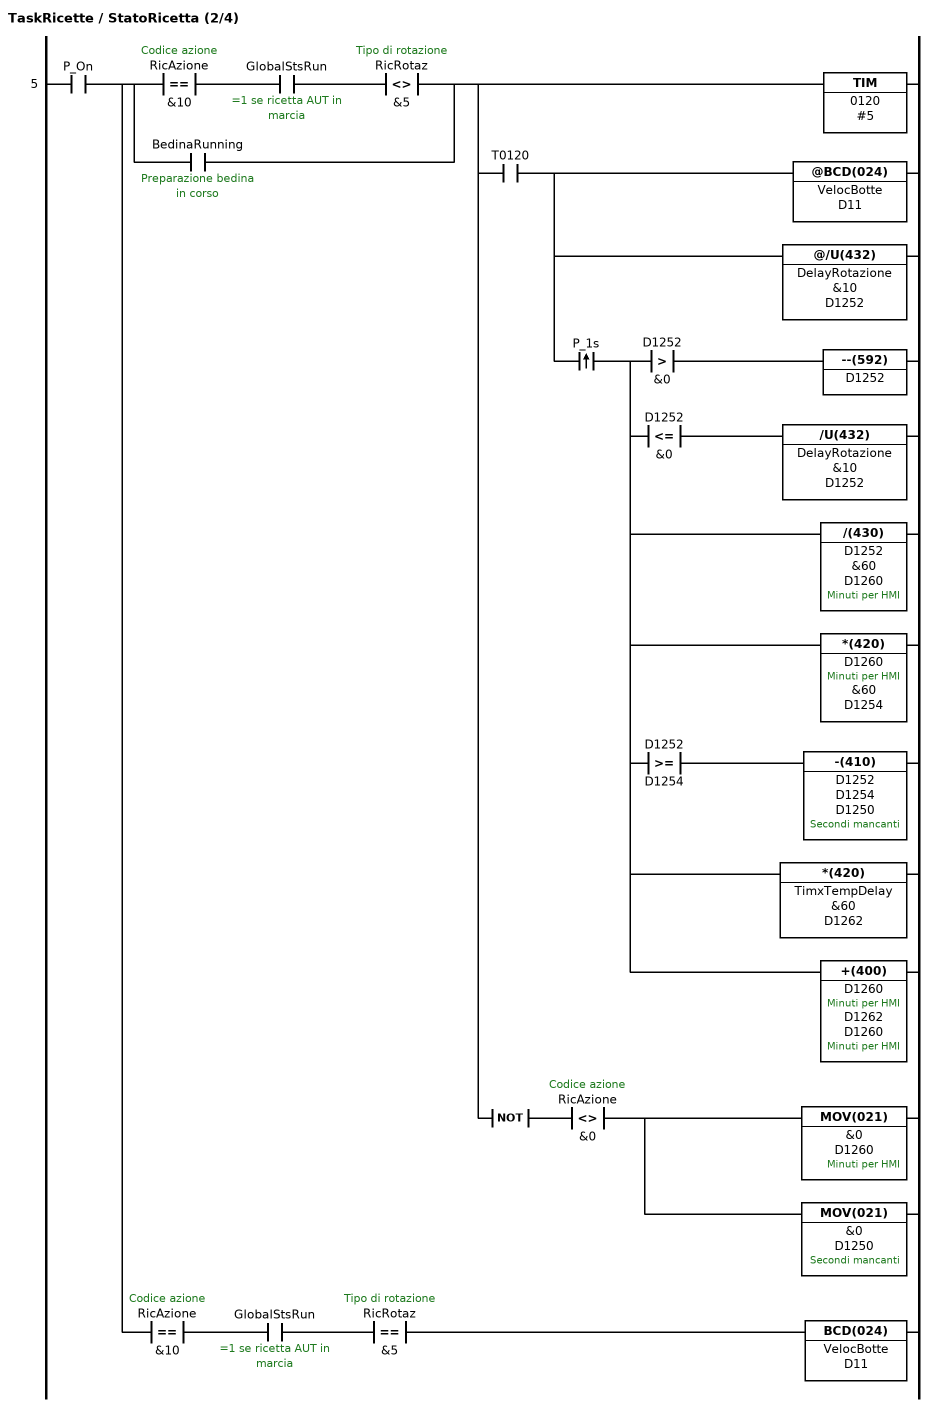
; [picture p48: TaskRicette / StatoRicetta, rungs 5-5]
; rung 5
LD P_On
OUT TR0
LD=(300) RicAzione &10  ; Codice azione
AND GlobalStsRun  ; =1 se ricetta AUT in marcia
AND<>(305) RicRotaz &5  ; Tipo di rotazione
OR BedinaRunning  ; Preparazione bedina in corso
ANDLD
OUT TR1
TIM 0120 #5
AND T0120
@BCD(024) VelocBotte D11
@/U(432) DelayRotazione &10 D1252
@AND P_1s
OUT TR2
AND>(320) D1252 &0
--(592) D1252
LD TR2
AND<=(315) D1252 &0
/U(432) DelayRotazione &10 D1252
LD TR2
/(430) D1252 &60 D1260  ; Minuti per HMI
*(420) D1260 &60 D1254  ; Minuti per HMI
AND>=(325) D1252 D1254
-(410) D1252 D1254 D1250  ; Secondi mancanti
LD TR2
*(420) TimxTempDelay &60 D1262
+(400) D1260 D1262 D1260  ; Minuti per HMI
LD TR1
NOT(520)
AND<>(305) RicAzione &0  ; Codice azione
MOV(021) &0 D1260  ; Minuti per HMI
MOV(021) &0 D1250  ; Secondi mancanti
LD TR0
AND=(300) RicAzione &10  ; Codice azione
AND GlobalStsRun  ; =1 se ricetta AUT in marcia
AND=(300) RicRotaz &5  ; Tipo di rotazione
BCD(024) VelocBotte D11

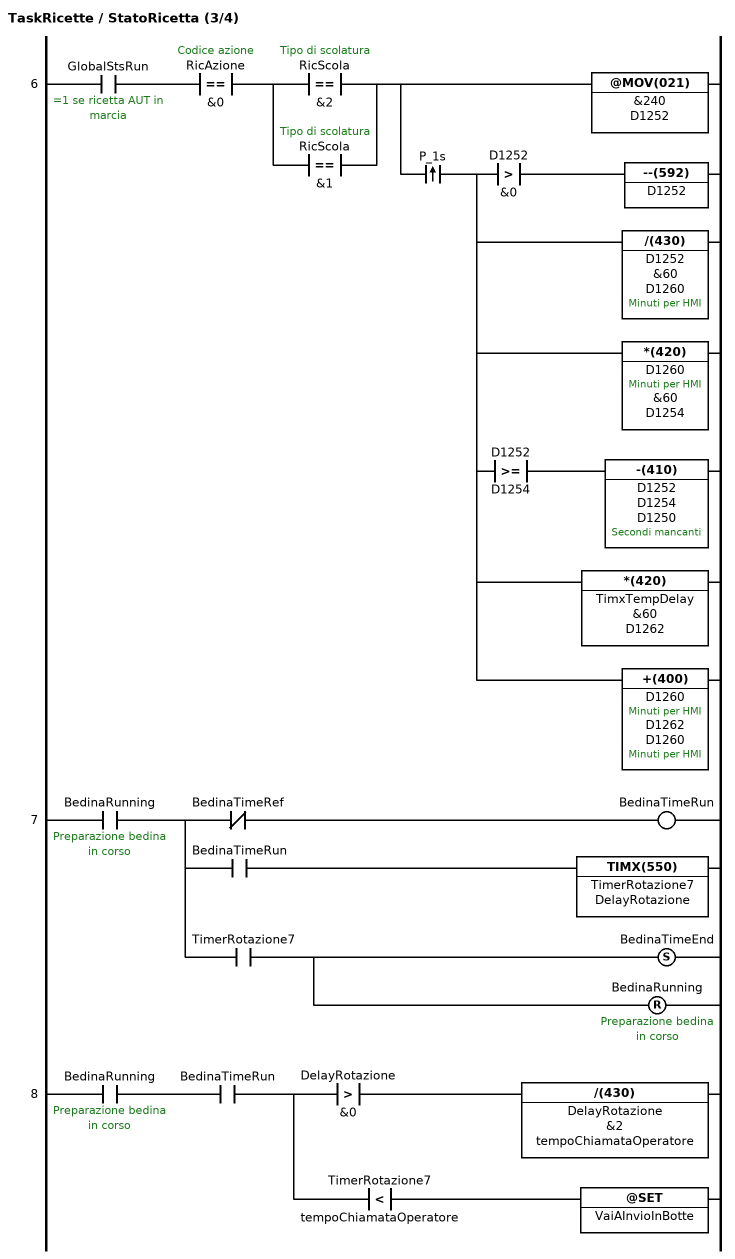
; rung 6
LD GlobalStsRun  ; =1 se ricetta AUT in marcia
AND=(300) RicAzione &0  ; Codice azione
LD=(300) RicScola &2  ; Tipo di scolatura
OR=(300) RicScola &1  ; Tipo di scolatura
ANDLD
@MOV(021) &240 D1252
@AND P_1s
OUT TR0
AND>(320) D1252 &0
--(592) D1252
LD TR0
/(430) D1252 &60 D1260  ; Minuti per HMI
*(420) D1260 &60 D1254  ; Minuti per HMI
AND>=(325) D1252 D1254
-(410) D1252 D1254 D1250  ; Secondi mancanti
LD TR0
*(420) TimxTempDelay &60 D1262
+(400) D1260 D1262 D1260  ; Minuti per HMI
; rung 7
LD BedinaRunning  ; Preparazione bedina in corso
OUT TR0
ANDNOT BedinaTimeRef
OUT BedinaTimeRun
LD TR0
AND BedinaTimeRun
TIMX(550) TimerRotazione7 DelayRotazione
LD TR0
AND TimerRotazione7
SET BedinaTimeEnd
RSET BedinaRunning  ; Preparazione bedina in corso
; rung 8
LD BedinaRunning  ; Preparazione bedina in corso
AND BedinaTimeRun
OUT TR0
AND>(320) DelayRotazione &0
/(430) DelayRotazione &2 tempoChiamataOperatore
LD TR0
AND<(310) TimerRotazione7 tempoChiamataOperatore
@SET VaiAInvioInBotte

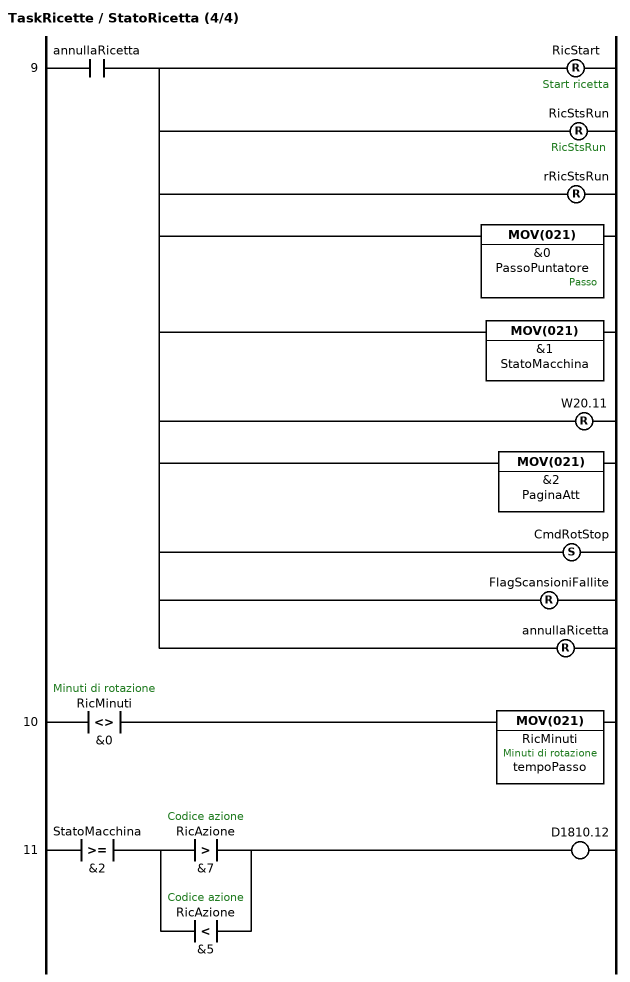
; rung 9
LD annullaRicetta
RSET RicStart  ; Start ricetta
RSET RicStsRun  ; RicStsRun
RSET rRicStsRun
MOV(021) &0 PassoPuntatore  ; Passo
MOV(021) &1 StatoMacchina
RSET W20.11
MOV(021) &2 PaginaAtt
SET CmdRotStop
RSET FlagScansioniFallite
RSET annullaRicetta
; rung 10
LD<>(305) RicMinuti &0  ; Minuti di rotazione
MOV(021) RicMinuti tempoPasso  ; Minuti di rotazione
; rung 11
LD>=(325) StatoMacchina &2
LD>(320) RicAzione &7  ; Codice azione
OR<(310) RicAzione &5  ; Codice azione
ANDLD
OUT D1810.12

### Section END

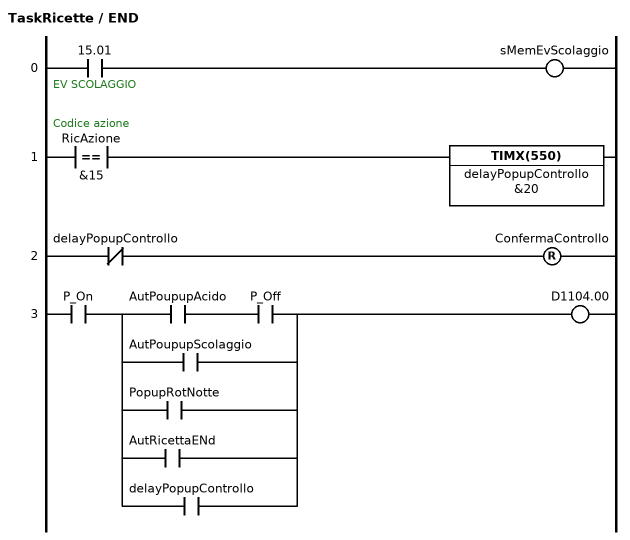
; rung 0
LD 15.01  ; EV SCOLAGGIO
OUT sMemEvScolaggio
; rung 1
LD=(300) RicAzione &15  ; Codice azione
TIMX(550) delayPopupControllo &20
; rung 2
LDNOT delayPopupControllo
RSET ConfermaControllo
; rung 3
LD P_On
LD AutPoupupAcido
AND P_Off
OR AutPoupupScolaggio
OR PopupRotNotte
OR AutRicettaENd
OR delayPopupControllo
ANDLD
OUT D1104.00
; rung 4
END(001)

## Program CicliStep (cyclic task 2)
Local symbols
CmdRst D2000.00 BOOL
CmdStart D2000.01 BOOL
Index D2010 INT
MemRiga D2012 WORD
StepCiclo D2001.00 BOOL[15]
StsEnd D2000.02 BOOL
StsRun D2000.03 BOOL
TempAnnoNecessario D2016 DINT
i D2014 INT
reset1 W20.10 BOOL
reset2 W20.11 BOOL
tempCondStep1 W20.12 BOOL
 IF TimerSaltaPasso.CF = TRUE  AND MemTimSkip=FALSE THEN
	Index:= 1;
	CmdRotAv:= false;
	CmdRotInd:= false;
	CmdRotAlt:= false;
	CmdRotStop:= false;
	CmdRotNotte:= false;
	CmdAcqua:= false;
	CmdFormico:= false;
	CmdGlutaral:= false;
	CmdScolaggioDecrementoAsse:= false;
	CmdScolaggioNormale:= false;
	PopupMancatoScolaggio:= false;
	RichiestaLetturaBarcode:= false;
	AutCmdNotturno:= false;
	AutPoupupScolaggio:= false;

end_if;
MemTimSkip:= TimerSaltaPasso.CF;
 
 (*Stop Riga*)
IF NOT  RicStart then
	StsRun:= false;
	(*StsEnd:= true;
	Index:= 5;*)
END_IF;
 
 
 (* Reset ciclo e comandi vari *)
IF CmdRst = TRUE THEN
	StsRun:= false;
	CmdStart:= false;
	CmdRst := false;	
END_IF;
GlobalGreenFlash:= false;
GlobalGreenLight:= false;
LetturaPesoREAL:= DINT_TO_REAL(LetturaPesoDINT);
		LetturaPesoREAL:= LetturaPesoREAL/1000,0;
		TolleranzaInf:= PesoNecessarioRicetta-((PesoNecessarioRicetta*Tolleranza)/100,0);
	(*I comandi da temperatura sono SET, vengono resettati dopo 1s sennò non li prende usando il momentaneo*)
TIMX(CmdTemperaturaON=true,TimerPIDon,10);
TIMX(CmdTemperaturaOFF=true,TimerPIDoff,10);
IF TimerPIDon.CF=TRUE THEN
	CmdTemperaturaON:= false;
END_IF;
IF TimerPIDoff.CF=TRUE THEN
	CmdTemperaturaOFF:= false;
END_IF;
(*Salvataggio ID riga per cambio riga*)
IF RicRigNum<>MemRiga THEN
	CmdStart:= true;
END_IF;
MemRiga:= RicRigNum;

(* Start riga *)
IF (CmdStart AND RicStsRun)= true THEN
	StsRun:= true;
	Index:= 1;
	CmdStart:= false;
	StsEnd:= false;
	FlagStsEnd:= false;
ELSIF RicStsRun=FALSE THEN
	StsRun:= false;
	Index:= 0;
END_IF;

FOR i:=0 TO 5 DO
	IF Index=i THEN	
		StepCiclo[i]:= true;
	ELSE
		StepCiclo[i]:= false;
	END_if;
END_FOR;

(* Cicli in base a codice azione *)
(* RIempimento acqua *)
IF RicAzione=5 THEN
	(* Passaggio parametri *)
	IF StepCiclo[1]=true THEN
		TemperaturaAcquaPerBCD:= INT_TO_WORD(((WORD_TO_INT(RicGradi)) * 10));
		LitriAcqua:= INT_TO_BCD_WORD(REAL_TO_INT(RicPeso/10,0));
		(*Controllo se è già stato eseguito un riempimento in precedenza*)
		IF FlagRiempimentoAcqua = TRUE THEN
			(*Riempimento già eseguito, richiedo la presenza operatore*)
			PopupMancatoScolaggio:= TRUE;
			IF PopupMancatoScolaggio=TRUE AND ConfermaMancatoScolaggio THEN (*Quando viene confermato il riempimento nonostante non ho scolaggio*)
				PopupMancatoScolaggio:= false;
				ConfermaMancatoScolaggio:= false;
				Index:= 2;
			END_IF;
		ELSE (*Se non è già avvenuto, proseguo*)		
			Index:= 2;
		end_if;
	END_IF;
	(*Comando*)
	IF StepCiclo[2]=true THEN
		CmdAcqua:= true;
		Index:= 3;
	END_IF;
	(* Attesa ritorno *)
	IF StepCiclo[3]=TRUE AND (FeedbackAcqua=TRUE OR (acqua_litriErogati >= (acqua_setpointRicetta/2))) THEN
		FlagRiempimentoAcqua:= TRUE;
		Index:= 4;
	END_IF;
	(* Attesa fine operazione *)
	(*IF StepCiclo[4]=true AND FeedbackAcqua=false THEN*)
	IF StepCiclo[4]=true AND (FeedbackAcqua=false OR (acqua_litriErogati >= (acqua_setpointRicetta/2)))  THEN
		TemperaturaMacchina:= TemperaturaAcqua;
		VelocBotte:= 9;
		CmdTemperaturaON:= true;
		IF NOT flagPrimoRiempimento then
			CmdRotAv:= true;
			IF FeedbackRotAv=TRUE then
				CmdRotAv:= FALSE;
				flagPrimoRiempimento := true;
				StsRun:= false;
				StsEnd:= true;			
			end_if;
		ELSIF flagPrimoRiempimento THEN
			StsRun:= false;
			StsEnd:= true;	
		end_if;		
	END_IF;
END_IF;

(* RIempimento formico *)
IF RicAzione=6 THEN
	(* Passaggio parametri *)
	tempCondStep1:= StepCiclo[1]=true  AND presenzaOpAcido=FALSE AND VaiAInvioInBotte=TRUE;
	TIMX(tempCondStep1,TimerFormico1,20);
	TIMX(TimerFormico1.CF,TimerFormico2,40);
	TIMX(StepCiclo[2]=true,TimerFormico3,20);
	TIMX(StepCiclo[2]=true,TimerFormico4,40);
	TIMX(StepCiclo[3]=true,TimerFormico5,20);
	TIMX(StepCiclo[3]=true,TimerFormico6,40);
	IF StepCiclo[1]=true THEN
		AutPoupupTBedina:= 1;
		PesoFormico:=  INT_TO_BCD_WORD(REAL_TO_INT(RicPeso*10,0));
		(*AutPoupupAcido:= TRUE;
		IF presenzaOpAcido=TRUE THEN
			presenzaOpAcido:= FALSE;*)
		IF VaiAInvioInBotte=TRUE AND presenzaOpAcido=FALSE THEN															(*attesa metà rotazione*)
			RichiestaFormico:= true;
			IF TimerFormico1.CF=TRUE THEN
				RichiestaFormico:= false;
				IF TimerFormico2.CF=TRUE THEN
					Index:= 2;
				END_IF;
			END_IF;
		END_IF;
	end_if;
	(*Comando*)
	IF StepCiclo[2]=true THEN
		SceltaFormico:= true;
		IF TimerFormico3.CF=TRUE THEN
			SceltaFormico:= false;
			IF TimerFormico4.CF=TRUE THEN
			Index:= 3;
			END_IF;
		END_IF;
	END_IF;
	(* Attesa ritorno *)
	IF StepCiclo[3] =true THEN
		CmdFormico:= true;
		IF TimerFormico5.CF=TRUE THEN
			CmdFormico:= false;
			
			IF TimerFormico6.CF=TRUE AND FeedbackFormico=TRUE THEN
				(*AutPoupupAcido:= true;
				confermaVaiABedina:= true;
				Index:= 4;*)
				Index:= 5;
			END_IF;
				END_IF;
	END_IF;
	(* Attesa fine operazione *)
	IF StepCiclo[4]=true AND AutPoupupAcido=false AND FeedbackFormico=false THEN
		AutPoupupTBedina:= 0;
		confermaVaiABedina:= false;
		IF confermaVaiABedina=FALSE then
			StsRun:= false;
			StsEnd:= true;
		end_if;
	END_IF;
	IF StepCiclo[5]=TRUE AND FeedbackFormico=false THEN
		AutPoupupAcido:= true;
		confermaVaiABedina:= true;
		IF AutPoupupAcido = TRUE then
			Index := 4;
		end_if;
	end_if;
	IF StepCiclo[4] = TRUE OR StepCiclo[5] = TRUE THEN
		visualizzaKgAcido := TRUE;
	ELSE
		visualizzaKgAcido:= FALSE;
	end_If;
END_IF;

(* RIempimento glutaraldeide *)
IF RicAzione=7 THEN
	(* Passaggio parametri *)
	TIMX(StepCiclo[1]=true,TimerGlutar1,20);
	TIMX(StepCiclo[1]=true,TimerGlutar2,40);
	TIMX(StepCiclo[2]=true,TimerGlutar3,20);
	TIMX(StepCiclo[2]=true,TimerGlutar4,40);
	TIMX(StepCiclo[3]=true,TimerGlutar5,20);
	TIMX(StepCiclo[3]=true,TimerGlutar6,40);
	IF StepCiclo[1]=true THEN
		AutPoupupTBedina:= 1;
		PesoGlutaral:=  INT_TO_BCD_WORD(REAL_TO_INT(RicPeso*10,0));
		AutPoupupAcido:= TRUE;
		IF presenzaOpAcido=TRUE THEN
			presenzaOpAcido:= FALSE;
			SceltaGlutar:= true;
			IF TimerGlutar1.CF=TRUE THEN
				SceltaGlutar:= false;
				IF TimerGlutar2.CF=TRUE THEN
					Index:= 2;
				END_IF;
			END_IF;
		end_if;
	END_IF;
	(*Comando*)
	IF StepCiclo[2]=true THEN
		RichiestaGlutar:= true;
		IF TimerGlutar3.CF=TRUE THEN
			RichiestaGlutar:= false;
			IF TimerGlutar4.CF=TRUE THEN
			Index:= 3;
			END_IF;
		END_IF;
	END_IF;
	(* Attesa ritorno *)
	IF StepCiclo[3] =true THEN
		CmdGlutaral:= true;
		IF TimerGlutar5.CF=TRUE THEN
			CmdGlutaral:= false;
			IF TimerGlutar6.CF=TRUE AND FeedbackGlutaral=TRUE THEN
				(*AutPoupupAcido:= true;
				Index:= 4;*)
				Index:= 5;
			END_IF;
				END_IF;
	END_IF;
	(* Attesa fine operazione *)
	IF StepCiclo[4]=true AND AutPoupupAcido=false AND FeedbackGlutaral=false THEN
		AutPoupupTBedina:= 0;
		confermaVaiABedina:= false;
		IF confermaVaiABedina=FALSE THEN
			StsRun:= false;
			StsEnd:= true;
		end_if;
	END_IF;
	IF StepCiclo[5]=TRUE AND FeedbackFormico=FALSE THEN
		AutPoupupAcido:=TRUE;
		confermaVaiABedina:=TRUE;
		IF AutPoupupAcido=TRUE THEN
			Index:= 4;
		end_if;
	END_IF;
	
	IF StepCiclo[4]=TRUE OR StepCiclo[5]=TRUE THEN
		visualizzaKgGlutaral:= TRUE;
	ELSE
		visualizzaKgGlutaral:= FALSE;
	END_IF;
END_IF;

(* Aggiorna temperatura macchina in rotazione *)
IF RicAzione=10 THEN
	IF RicGradi <> 0 then
		TemperaturaMacchina :=  INT_TO_BCD_WORD(((WORD_TO_INT(RicGradi)) * 10));
	ELSE
		TemperaturaMacchina := 10;
	end_if;
end_if;


(* Rotazione avanti, tipo 1 *)
IF RicAzione=10 AND RicRotaz=1 THEN
	(* Passaggio parametri *)
	IF StepCiclo[1]=true THEN
		VelocBotte:= INT_TO_WORD(REAL_TO_INT((INT_TO_REAL(WORD_TO_INT(RicSpeed))) * 1,24));
		Index:= 2;
	END_IF;
	(*Comando*)
	IF StepCiclo[2]=true THEN
		CmdRotAv:= true;
		Index:= 3;
	END_IF;
	(* Attesa ritorno *)
	IF StepCiclo[3]=true AND FeedbackRotAv=true THEN
		TIMX(StepCiclo[3]=true,TimerRotazione,DelayRotazione);
		CmdRotAv:= false;
		IF TimerRotazione.CF THEN		
			Index:= 4;
		END_IF;
	END_IF;
	(* Attesa fine operazione *)
	IF StepCiclo[4]=true  THEN	
		StsRun:= false;
		StsEnd:= true;
	END_IF;
END_IF;

(* Rotazione indietro, tipo 2 *)
IF RicAzione=10 AND RicRotaz=2 THEN
	(* Passaggio parametri *)
	IF StepCiclo[1]=true THEN
		VelocBotte:= INT_TO_WORD(REAL_TO_INT((INT_TO_REAL(WORD_TO_INT(RicSpeed))) * 1,24));
		Index:= 2;
	END_IF;
	(*Comando*)
	IF StepCiclo[2]=true THEN
		CmdRotInd:= true;
		Index:= 3;
	END_IF;
	(* Attesa ritorno *)
	IF StepCiclo[3]=true AND FeedbackRotInd=true THEN
		TIMX(StepCiclo[3]=true,TimerRotazione,DelayRotazione);
		CmdRotInd:= false;
		IF TimerRotazione.CF THEN		
			Index:= 4;
		END_IF;
	END_IF;
	(* Attesa fine operazione *)
	IF StepCiclo[4]=true  THEN	
		StsRun:= false;
		StsEnd:= true;
	END_IF;
END_IF;

(* Rotazione alternata, tipo 3 *)
IF RicAzione=10 AND RicRotaz=3 THEN
	(* Passaggio parametri *)
	IF StepCiclo[1]=true THEN
		VelocBotte:= INT_TO_WORD(REAL_TO_INT((INT_TO_REAL(WORD_TO_INT(RicSpeed))) * 1,24));
		IF RicMinuti<=60 then
			DelayRotazione:= (WORD_TO_UINT(RicMinuti)*600);
			TimxTempDelay:= 0;
		ELSIF RicMinuti>60 THEN
			TimxTempDelay:= 0;
			TimxRicMinuti:= WORD_TO_INT(RicMinuti);
			WHILE TimxRicMinuti>60 DO
				TimxRicMinuti:= TimxRicMinuti-60;
				TimxTempDelay:= TimxTempDelay+1;
			END_WHILE;
			DelayRotazione:= (INT_TO_UINT(TimxRicMinuti))*600;
		end_if;
		Index:= 2;
		CmdRotAlt:= true;
	END_IF;
	(*Comando*)
	TIMX(StepCiclo[2]=TRUE,timerRotazioneStep2, 10);
	IF StepCiclo[2]=true AND timerRotazioneStep2.CF = TRUE THEN
		Index:= 3;
	END_IF;
	(* Attesa ritorno *)
	IF TimxTempDelay= 0 then
		TIMX(StepCiclo[3]=true,TimerRotazione3,DelayRotazione);
	ELSIF TimxTempDelay>0 THEN
		TIMX(StepCiclo[3]=true,TimerRotazione3,36000);
	end_if;
	IF StepCiclo[3]=true AND FeedbackRotAlt=true THEN
		CmdRotAlt:= false;
		IF TimerRotazione3.CF THEN
				IF TimxTempDelay= 0 then
					Index:= 4;
				ELSIF TimxTempDelay>0 THEN
					TimxTempDelay:=TimxTempDelay-1;
					Index:= 2;
				end_if;
		END_IF;
	END_IF;
	(* Attesa fine operazione *)
	IF StepCiclo[4]=true  THEN	
		StsRun:= false;
		StsEnd:= true;
	END_IF;
END_IF;

(* Ferma rotazione, tipo 4 *)
IF RicAzione=10 AND RicRotaz=4 THEN
	(* Passaggio parametri *)
	IF StepCiclo[1]=true THEN
		Index:= 2;
	END_IF;
	(*Comando*)
	IF StepCiclo[2]=true THEN
		CmdRotStop:= true;
		Index:= 3;
	END_IF;
	(* Attesa ritorno *)
	TIMX(StepCiclo[3]=true,TimerRotazione4,100);
	IF StepCiclo[3]=true THEN
		IF TimerRotazione4.CF THEN		
			CmdRotStop:= FALSE;
			Index:= 4;
		END_IF;
	END_IF;
	(* Attesa fine operazione *)
	IF StepCiclo[4]=true  THEN	
		StsRun:= false;
		StsEnd:= true;
	END_IF;
END_IF;

(* Rotazione alternata notte, tipo 5 *)
IF RicAzione=10 AND RicRotaz=5 THEN
	(* Passaggio parametri *)
	IF StepCiclo[1]=true THEN
		PopupRotNotte:= false;
		VelocBotte:= 6;
		OreAltPreNotte:= 0;
		MinAltPreNotte:= 5;
		Index:= 2;
	END_IF;
	(*Comando*)
	IF StepCiclo[2]=true THEN
		AutCmdNotturno:= TRUE;
		Index:= 3;
	END_IF;
	(* Attesa ritorno *)
	IF StepCiclo[3]=true AND FeedbackRotAlt=true THEN
			PopupRotNotte:= true;
			Index:= 4;
		END_IF;
	END_IF;
	(* Attesa fine operazione *)
	IF StepCiclo[4]=true AND ConfermaRotNotte=true  THEN
		PopupRotNotte:= false;
		StsRun:= false;
		StsEnd:= true;
	END_IF;

(* Rotazione alternata, tipo 7 *)
IF RicAzione=10 AND RicRotaz=7 THEN
	(* Passaggio parametri *)
	IF StepCiclo[1]=true THEN
		BedinaTimeEnd:= FALSE;
		VelocBotte:= INT_TO_WORD(REAL_TO_INT((INT_TO_REAL(WORD_TO_INT(RicSpeed))) * 1,24));
		IF RicMinuti<=60 then
			DelayRotazione:= (WORD_TO_UINT(RicMinuti)*600);
			TimxBedinaDelay:= 0;
		ELSIF RicMinuti>60 THEN
			TimxBedinaDelay:= 0;
			TimxRicMinuti:= WORD_TO_INT(RicMinuti);
			WHILE TimxRicMinuti>60 DO
				TimxRicMinuti:= TimxRicMinuti-60;
				TimxBedinaDelay:= TimxBedinaDelay+1;
			END_WHILE;
			DelayRotazione:= (INT_TO_UINT(TimxRicMinuti))*600;
		end_if;
		Index:= 2;
		CmdRotAlt:= true;
		BedinaRunning:= true;
	END_IF;
	(*Comando*)
	IF StepCiclo[2]=true THEN
		Index:= 3;
	END_IF;
	
	IF StepCiclo[3]=true AND FeedbackRotAlt=true THEN
		CmdRotAlt:= false;
		AutPupupInvioBotte:= FALSE;
	    Index:= 4;
	END_IF;
	(* Attesa fine operazione *)
	IF StepCiclo[4]=true  THEN	
		StsRun:= false;
		StsEnd:= true;
		(*BedinaRunning:= FALSE;*)
	END_IF;
END_IF;

(* Preparazione bedina, tipo 7  *)
IF RicAzione=50 AND RicRotaz=7 THEN
	(* Passaggio parametri *)
	IF StepCiclo[1]=true THEN
		(*VaiAInvioInBotte:= TRUE;*)
		RichiestaLetturaBarcode:= TRUE;
		AutPoupupBedina:= 1;
		AutPoupupTBedina:= 1;
		FlagAbilitaScansioni:= TRUE;
	        	
				FlagScansioniFallite:= FALSE;
				FlagIgnoraScansioniFallite:= FALSE;
				NumeroScansioni:= 0;
				FlagRitentaScansioni:= FALSE;
				StatoScansione:= 0;
		Index:= 2;
	END_IF;
	(*Comando*)
	IF StepCiclo[2]=true AND ((LetturaPesoREAL=0,0) AND LetturaCodPro=0 AND LetturaRicetta=0) THEN
		ProdottoErratoPopup:= false;
		StatoScansione:= 1;
		Index:= 3;
	END_IF;
	(* Attesa ritorno *)

	IF StepCiclo[3]=true AND (FlagScansioniFallite=FALSE) AND (LetturaPesoREAL<>0,0) AND (LetturaCodPro<>0) AND (LetturaRicetta<>0) THEN
		(*Conversione peso da DINT da bilanca a reale, in Kg. Calcolo tolleranze da parametro tolleranza % (5%, per ora)*)
		LetturaPesoREAL:= DINT_TO_REAL(LetturaPesoDINT);
		LetturaPesoREAL:= LetturaPesoREAL/REAL1000;
		TolleranzaInf:= PesoNecessarioRicetta-((PesoNecessarioRicetta*Tolleranza)/PercentualeREAL);
		TolleranzaSup:= PesoNecessarioRicetta+((PesoNecessarioRicetta*Tolleranza)/PercentualeREAL);
		(*Su codice a barre Anno e n°Ricetta sono un codice unico, vengono uniti in quanto separati*)
		TempAnnoNecessario:= INT_TO_DINT(AnnoNecessarioRicetta);
		LetturaRicettaTemp:= (TempAnnoNecessario*10000000)+(RicettaNecessariaRicetta);
		
						
		(*Controlla corrispondeza peso, codice prodotto, codice ricetta*)
			IF LetturaPesoREAL>TolleranzaInf AND LetturaPesoREAL<TolleranzaSup AND LetturaCodPro= CodiceNecessarioRicetta AND LetturaRicetta=LetturaRicettaTemp then		
				Index:= 4;
				FlagNuovaScansione:= false;
				RichiestaLetturaBarcode:= FALSE;
				AutPoupupBedina:= 0;
				AutPoupupTBedina:= 0;
				FlagAbilitaScansioni:= FALSE;
				NumeroScansioni:= 0;
				ELSE
				(*Se il prodotto non è giusto, segno 1 tentativo e resetto tutto*)
				StatoScansione:= 2;
				
				IF NumeroScansioni<2 THEN
					NumeroScansioni:= NumeroScansioni+1;
					Index:= 2;
				
				ELSIF NumeroScansioni>=2 THEN
					FlagScansioniFallite:= TRUE;
									
				END_IF;;
		
		FlagNascondiTasti:= NOT(FlagScansioniFallite OR RichiestaLetturaBarcode);
	END_IF;
				
END_IF;		
	(* Attesa fine operazione *)
		IF StepCiclo[3]=true AND FlagScansioniFallite=TRUE THEN
			AutPoupupBedina:= 0;
			IF FlagIgnoraScansioniFallite=TRUE THEN
				FlagScansioniFallite:= FALSE;
				FlagIgnoraScansioniFallite:= FALSE;
				RichiestaLetturaBarcode:= FALSE;
			    AutPoupupBedina:= 0;
				NumeroScansioni:= 0;
				Index:= 4;
			END_IF;
		END_IF;		
	(*invio in bedina manuale completato, conferma da operatore*)
	IF StepCiclo[4]=true  THEN
		
		ConfermaBedina:= False;
		RichiestaConfermaBedina:= false;
		StsRun:= false;
		StsEnd:= true;
				
	END_IF;
END_IF;

(* Invio in botte, tipo 8 *)
IF RicAzione=10 AND RicRotaz=8 THEN
	IF StepCiclo[1]=true AND BedinaTimeEnd=FALSE THEN
	AutPoupupTBedina:= 1;
	END_IF;
	(* Passaggio parametri *)
	IF StepCiclo[1]=true AND BedinaTimeEnd=TRUE THEN
		IF FlagSolido=TRUE THEN
			CmdRotStop:= true;
		end_if;
		Index:= 2;
		AutPoupupTBedina:= 0;
		BedinaTimeEnd:= FALSE;
	END_IF;
	(*Comando*)
	TIMX(StepCiclo[2]=true,TimerRotazione4,100);
	IF StepCiclo[2]=true THEN
		IF FlagSolido=TRUE THEN
			IF TimerRotazione4.CF THEN		
				CmdRotStop:= FALSE;
				Index:= 3;
				FlagSolido:= false;
				(*VaiAInvioInBotte:= true;*)
			END_IF;
		ELSE
			Index:= 3;
			(*VaiAInvioInBotte:= true;*)
		end_if;
	END_IF;
	(* Attesa ritorno *)
	IF StepCiclo[3]=true THEN
		AutPupupInvioBotte:= true;
			Index:= 4;
		(*END_IF;*)
	END_IF;
	(* Attesa fine operazione *)
	IF invioConRisciacquoON OR invioSenzaRisciacquoON THEN
		ConfermaInvioBotte:= FALSE;
	end_if;
	IF StepCiclo[4]=true AND ConfermaInvioBotte=true AND NOT invioConRisciacquoON AND NOT invioSenzaRisciacquoON THEN	
		ConfermaInvioBotte:= false;
		AutPupupInvioBotte:= false;
		StsRun:= false;
		StsEnd:= true;
	END_IF;
END_IF;

(* Controllo *)
IF RicAzione=15 THEN
	(* Passaggio parametri *)
	IF StepCiclo[1]=true THEN
		Index:= 2;
	END_IF;
	(*Comando*)
	IF StepCiclo[2]=true THEN
		Index:= 3;
	END_IF;
	(* Attesa ritorno *)
	IF StepCiclo[3]=true AND delayPopupControllo.CF=TRUE THEN
		Index:= 4;
	END_IF;
	(* Attesa fine operazione *)
	IF StepCiclo[4]=true AND ConfermaControllo=True AND delayPopupControllo.CF=TRUE THEN	
		ConfermaControllo:= false;
		StsRun:= false;
		StsEnd:= true;
	END_IF;
END_IF;

(*Scolaggio a decremento da asse*)
IF RicScola=2 AND RicAzione= 0 THEN
	IF StepCiclo[1]=TRUE THEN
		CmdScolaggioDecrementoAsse:= true;
		IF StsScolaggioDecrementoAsse=TRUE THEN
			CmdScolaggioDecrementoAsse:= false;
			Index:= 2;
		END_IF;
	END_IF;
	IF StepCiclo[2]=TRUE THEN
		IF AutCmdStop=TRUE THEN
			FlagRiempimentoAcqua:= false;
			StsRun:= false;
			StsEnd:= true;
			flagPrimoRiempimento :=  FALSE;
		END_IF;
	END_IF;
(*ELSIF RicScola=1 AND RicAzione= 0 THEN
	IF StepCiclo[1]=TRUE THEN
		CmdScolaggioNormale:= true;
		TIMX(StepCiclo[1],TimerScolaggioON,10);
		IF TimerScolaggioON.CF=TRUE THEN
			CmdScolaggioNormale:= false;
			Index:= 2;
		END_IF;
	END_IF;
	IF StepCiclo[2]=TRUE THEN
		IF StsScolaggioNormale=FALSE THEN
			StsRun:= false;
			StsEnd:= true;
		END_IF;
	END_IF;*)
IF RicScola<>0 OR RicAzione=99 then
	CmdTemperaturaOFF:= true;
	TemperaturaMacchina:= 1;
end_if;
END_IF;	
TIMX((RicScola=1),TimerScolaggioNormale,2400);
IF RicScola=1 AND RicAzione= 0 THEN	
	IF TimerScolaggioNormale.CF = TRUE AND NOT flagFineScolaggio THEN
		AutPoupupScolaggio:= TRUE;
		flagFineScolaggio:= TRUE;
	END_IF;
	IF StepCiclo[1]=TRUE THEN
		CmdScolaggioNormale:= true;
		IF StsScolaggioNormale=TRUE THEN
			CmdScolaggioNormale:= false;
			Index:= 2;
		END_IF;
	END_IF;
	IF StepCiclo[2]=TRUE THEN
		IF AutCmdStop=TRUE THEN
			FlagRiempimentoAcqua:= false;
			StsRun:= false;
			StsEnd:= true;
			flagFineScolaggio:= FALSE;
			flagPrimoRiempimento :=  FALSE;
		END_IF;
	END_IF;
END_IF;	
(*Con la pausa non incremento il passo a fine azione*)
IF (NOT RicPause) AND RicStart then
	(* Cambio riga su fronte dello status end. Aumenta il puntatore e carica il passo successivo*)
	IF StsEnd<>FlagStsEnd THEN
		RicStato:=2;
		PassoPuntatoreINT:= WORD_TO_INT(PassoPuntatore);
		PassoPuntatoreINT:= (PassoPuntatoreINT+1);
		PassoPuntatore:= INT_TO_WORD(PassoPuntatoreINT);
		CaricaRIcetta:= true;
	END_IF;
	FlagStsEnd:= StsEnd;
ELSE
	StsRun:= false;
END_IF;

	
(*Copia  stsRun e comandi torretta luminosa in variabili globali*)
GlobalStsRun:= StsRun;
(*Se sono in marcia automatica, controllo torretta e stati in automatico, altrimenti sono esclusi*)
IF StsRun=TRUE then
	IF RicAzione=50 OR RicAzione=10 OR RicAzione=15 then
		CASE WORD_TO_INT(RicRotaz) OF
			1..7: (*Con rotazioni standard, luce fissa*)
				GlobalGreenLight:= true;
			(*7: Se invio in bedina o in botte, la luce lampeggia
				GlobalGreenFlash:= true;*)
		END_CASE;
	END_IF;
	(*Lampeggio torretta con conferma di mancato scolaggio*)
	IF (RicAzione=5 AND PopupMancatoScolaggio=TRUE) OR (RicAzione=10 AND  RicRotaz=8 AND BedinaRunning=FALSE) OR (RicAzione=15) (*OR (RicAzione=6)*)OR AutPoupupScolaggio= TRUE OR RicScola = 1 OR confermaVaiABedina=TRUE OR inserimentoProdottiRunning OR VaiAInvioInBotte THEN
		GlobalGreenFlash:= TRUE;
	END_IF;
    IF (RicAzione=10 AND  RicRotaz=8 AND BedinaRunning=TRUE) OR (RicAzione=0 AND RicScola=2 AND PopupMancatoScolaggio=false AND AutPoupupScolaggio= FALSE)  THEN
		GlobalGreenLight:= TRUE;
	END_IF;
	reset1:= FALSE;
ELSE
	(*Lo StsRun si reinizializza su ogni passo, attenzione alle memorie che vengono inserite di seguito*)
	(*Resetta memoria usate dalla ricetta*)
	IF reset1=FALSE then
	GlobalGreenLight:= false;
	GlobalGreenFlash:= false;
	RicAzione:= 0;
	RicRotaz:= 0;
	VisibilitàIndietroMan:= true;
	FlagRiempimentoAcqua:= false;
	CmdRotAv:= false;
	CmdRotInd:= false;
	CmdRotAlt:= false;
	IF stopDaBarriera = FALSE THEN
		CmdRotStop:= false;
	end_if;
	CmdRotNotte:= false;
	CmdAcqua:= false;
	CmdFormico:= false;
	CmdGlutaral:= false;
	CmdScolaggioDecrementoAsse:= false;
	CmdScolaggioNormale:= false;
	PopupMancatoScolaggio:= false;
	RichiestaLetturaBarcode:= false;
	AutCmdNotturno:= false;
	AutPupupInvioBotte:= false;
	AutPoupupBedina:= 0;
	AutPoupupTBedina:= 0;
	PopupRotNotte:= false;
	
	ConfermaInvioBotte:= false;
	AutPupupInvioBotte:= false;
	AutFlagConforme:= false;
	reset1:= TRUE;
	end_if;
END_IF;
IF rRicStsRun= FALSE AND NOT stopDaBarriera THEN
	IF reset2= FALSE then
	GlobalGreenLight:= false;
	GlobalGreenFlash:= false;
	RicAzione:= 0;
	RicRotaz:= 0;
	VisibilitàIndietroMan:= true;
	FlagRiempimentoAcqua:= false;
	CmdRotAv:= false;
	CmdRotInd:= false;
	CmdRotAlt:= false;
	CmdRotStop:= false;
	CmdRotNotte:= false;
	CmdAcqua:= false;
	CmdFormico:= false;
	CmdGlutaral:= false;
	CmdScolaggioDecrementoAsse:= false;
	CmdScolaggioNormale:= false;
	PopupMancatoScolaggio:= false;
	RichiestaLetturaBarcode:= false;
	AutCmdNotturno:= false;
	AutPupupInvioBotte:= false;
	AutPoupupBedina:= 0;
	AutPoupupTBedina:= 0;
	PopupRotNotte:= false;
				confermaVaiABedina:= false;
				flagFineScolaggio:= false;
				presenzaOpAcido:= false;
				inserimentoProdottiRunning:= false;
				AutPoupupTBedina:= 0;
				BedinaTimeEnd:= FALSE;
		
				FlagNuovaScansione:= false;
				RichiestaLetturaBarcode:= FALSE;
				AutPoupupBedina:= 0;
				FlagAbilitaScansioni:= FALSE;
				NumeroScansioni:= 0;
				
				ConfermaInvioBotte:= false;
				AutPupupInvioBotte:= false;
				AutFlagConforme:= false;
				
				reset2:= true;
	END_IF;
ELSE
	reset2:= false;
END_IF;
	(*Lampeggio torretta con fine ricetta*)
	IF AutRicettaENd=TRUE OR RicAzione=99 THEN
		GlobalGreenFlash:= TRUE;
	END_IF;
	
VisibilitàIndietroMan:= true;

(*(*Gestione stato della botte per supervisione*)
IF (StatoMacchina= 0) AND (PaginaAtt=2 OR PaginaAtt=13) AND RicStsRun= false THEN
	StatoMacchina:= 1;
ELSIF (PaginaAtt<>2) AND (StatoMacchina)<2 THEN
	StatoMacchina:= 0;
end_if;
IF (StatoMacchina=2 AND RicStsRun=TRUE) OR GlobalGreenLight=TRUE THEN
	StatoMacchina:= 3;
END_IF;
IF RicPause THEN
	StatoMacchina:= 4;
END_IF;
IF GlobalGreenFlash=TRUE THEN
	StatoMacchina:= 5;
END_IF;
IF RicAzione=99 THEN
	StatoMacchina:= 10;
end_if;
IF StatoMacchina=11 THEN
	StatoMacchina:= 0;
end_if;

luceProdotti:= FALSE;

IF delayAlternataOn = TRUE THEN
	CmdRotAlt := TRUE;
end_if;

## Program mgrRegistraDati (cyclic task 3)
Local symbols
cmdAnnullaRicetta D1810.11 BOOL  ; Comado di annullamento ricetta da HMI
indexScrittura D2511 INT
indexSottorigaAtt D2510 WORD
nuovaSottorigaReq D1810.13 BOOL
primaSottoriga E20000 INT
puntaRigaAtt E15001 INT
puntaSottorigaAtt E15000 INT
rigaInLavorazione D8000 INT
rigaTemporanea E15500 INT
sottorigaInRegistrazione D1811.00 BOOL
sottorigaInScrittura D1810.15 BOOL
statoRicetta D900 INT  ; se >0, ricetta in run
tempOreRotaz E15002 INT
tempPeso E15004 INT
tempSotAzione E15506 WORD  ; Codice azione
tempSotGradi E15564 WORD  ; Temperatura acqua
tempSotMinuti E15566 WORD  ; Minuti di rotazione
tempSotPeso E15560 REAL  ; Peso prodotto in Kg
tempSotRotaz E15568 WORD  ; Tipo di rotazione
tempSotScola E15570 WORD  ; Tipo di scolatura
tempSotSpeed E15572 WORD  ; Velocità (da 2 a 8)
tempSotStato E15588 WORD

### Section registrazioneSottoriga

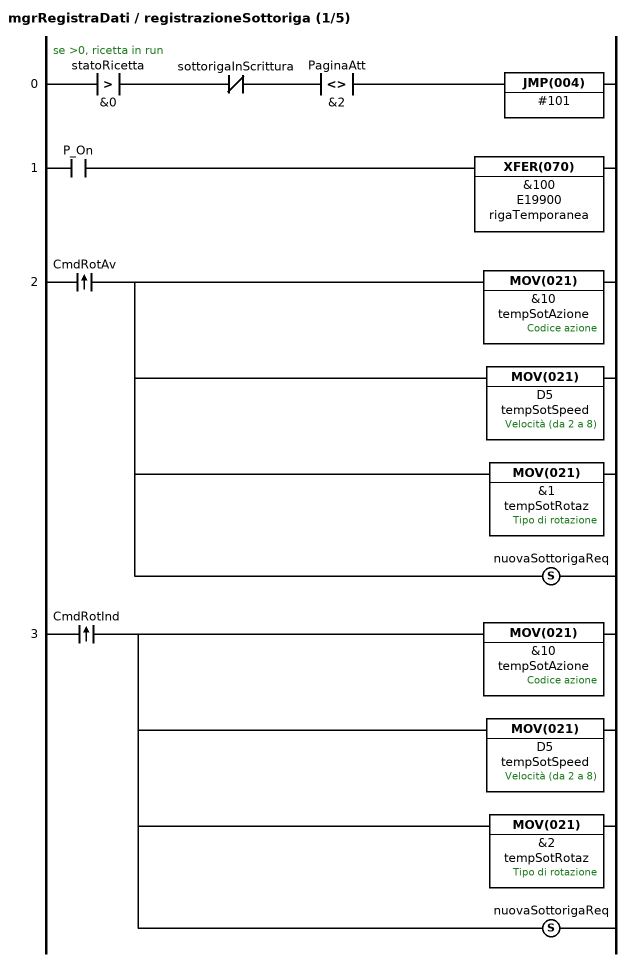
; rung 0
LD>(320) statoRicetta &0  ; se >0, ricetta in run
ANDNOT sottorigaInScrittura
AND<>(305) PaginaAtt &2
JMP(004) #101
; rung 1
LD P_On
XFER(070) &100 E19900 rigaTemporanea
; rung 2
@LD CmdRotAv
MOV(021) &10 tempSotAzione  ; Codice azione
MOV(021) D5 tempSotSpeed  ; Velocità (da 2 a 8)
MOV(021) &1 tempSotRotaz  ; Tipo di rotazione
SET nuovaSottorigaReq
; rung 3
@LD CmdRotInd
MOV(021) &10 tempSotAzione  ; Codice azione
MOV(021) D5 tempSotSpeed  ; Velocità (da 2 a 8)
MOV(021) &2 tempSotRotaz  ; Tipo di rotazione
SET nuovaSottorigaReq

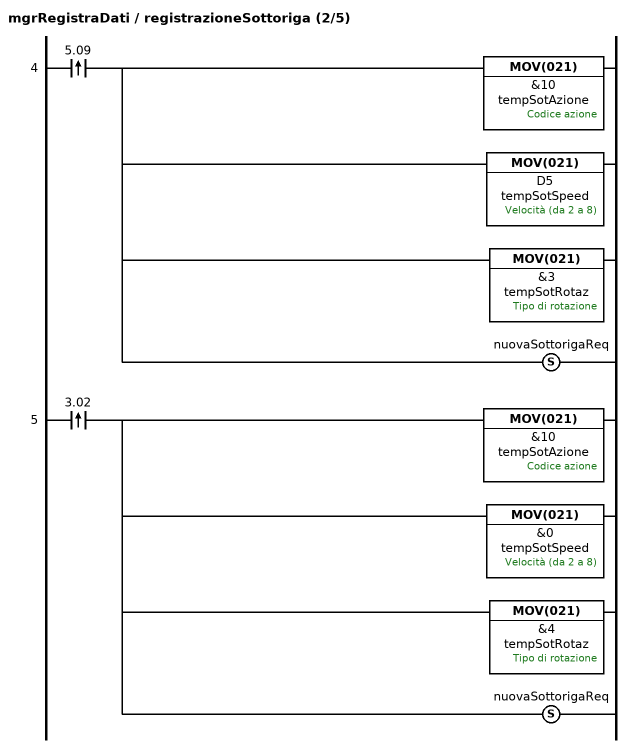
; rung 4
@LD 5.09
MOV(021) &10 tempSotAzione  ; Codice azione
MOV(021) D5 tempSotSpeed  ; Velocità (da 2 a 8)
MOV(021) &3 tempSotRotaz  ; Tipo di rotazione
SET nuovaSottorigaReq
; rung 5
@LD 3.02
MOV(021) &10 tempSotAzione  ; Codice azione
MOV(021) &0 tempSotSpeed  ; Velocità (da 2 a 8)
MOV(021) &4 tempSotRotaz  ; Tipo di rotazione
SET nuovaSottorigaReq

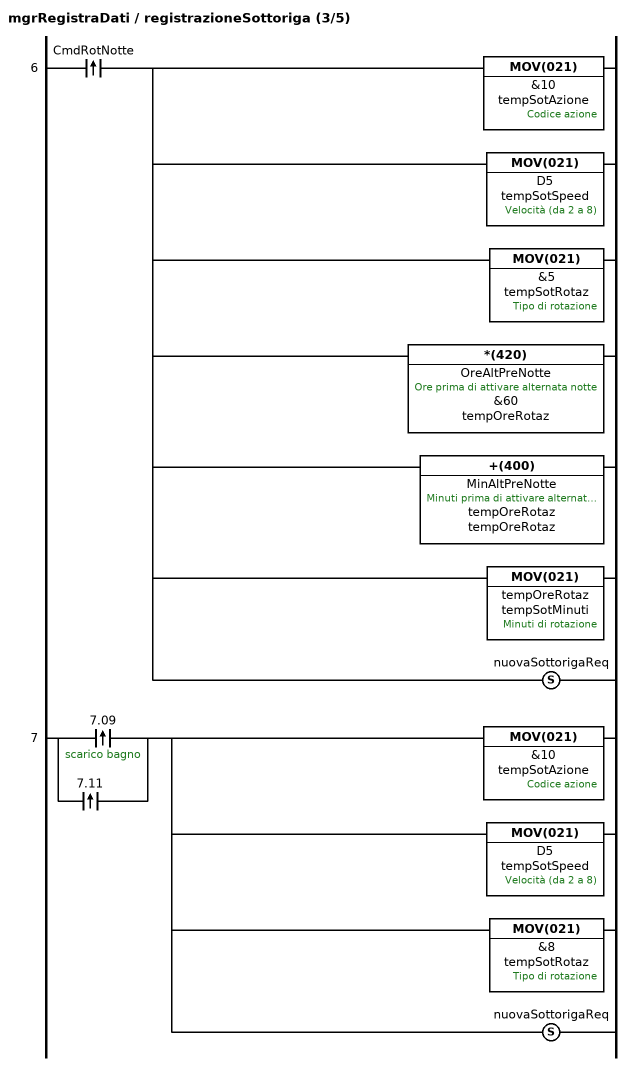
; rung 6
@LD CmdRotNotte
MOV(021) &10 tempSotAzione  ; Codice azione
MOV(021) D5 tempSotSpeed  ; Velocità (da 2 a 8)
MOV(021) &5 tempSotRotaz  ; Tipo di rotazione
*(420) OreAltPreNotte &60 tempOreRotaz  ; Ore prima di attivare alternata notte
+(400) MinAltPreNotte tempOreRotaz tempOreRotaz  ; Minuti prima di attivare alternata notte
MOV(021) tempOreRotaz tempSotMinuti  ; Minuti di rotazione
SET nuovaSottorigaReq
; rung 7
@LD 7.09  ; scarico bagno
@OR 7.11
MOV(021) &10 tempSotAzione  ; Codice azione
MOV(021) D5 tempSotSpeed  ; Velocità (da 2 a 8)
MOV(021) &8 tempSotRotaz  ; Tipo di rotazione
SET nuovaSottorigaReq

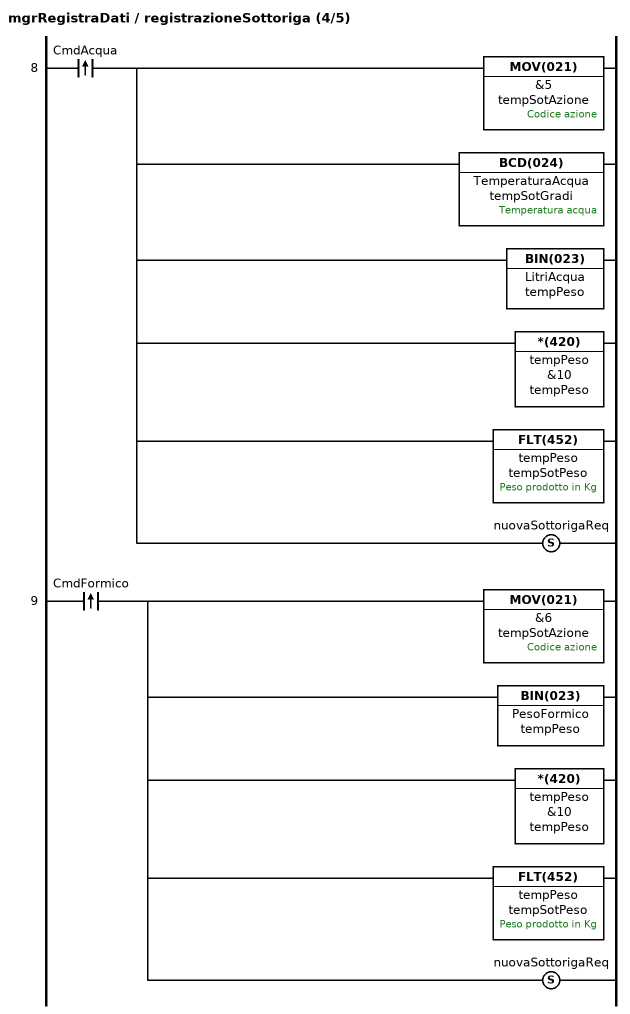
; rung 8
@LD CmdAcqua
MOV(021) &5 tempSotAzione  ; Codice azione
BCD(024) TemperaturaAcqua tempSotGradi  ; Temperatura acqua
BIN(023) LitriAcqua tempPeso
*(420) tempPeso &10 tempPeso
FLT(452) tempPeso tempSotPeso  ; Peso prodotto in Kg
SET nuovaSottorigaReq
; rung 9
@LD CmdFormico
MOV(021) &6 tempSotAzione  ; Codice azione
BIN(023) PesoFormico tempPeso
*(420) tempPeso &10 tempPeso
FLT(452) tempPeso tempSotPeso  ; Peso prodotto in Kg
SET nuovaSottorigaReq

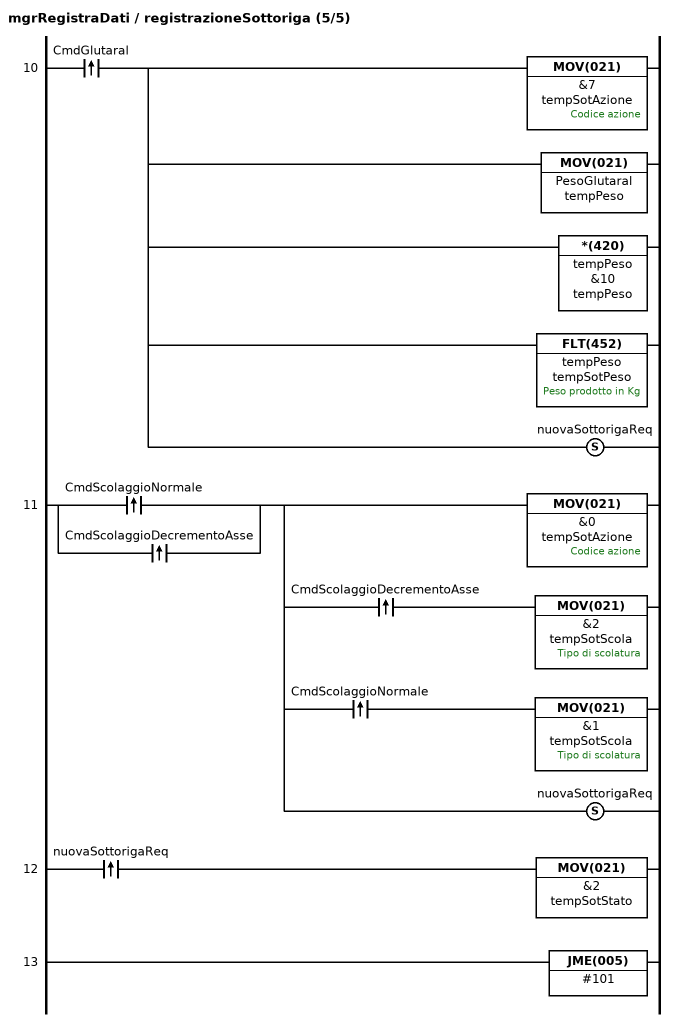
; rung 10
@LD CmdGlutaral
MOV(021) &7 tempSotAzione  ; Codice azione
MOV(021) PesoGlutaral tempPeso
*(420) tempPeso &10 tempPeso
FLT(452) tempPeso tempSotPeso  ; Peso prodotto in Kg
SET nuovaSottorigaReq
; rung 11
@LD CmdScolaggioNormale
@OR CmdScolaggioDecrementoAsse
OUT TR0
MOV(021) &0 tempSotAzione  ; Codice azione
@AND CmdScolaggioDecrementoAsse
MOV(021) &2 tempSotScola  ; Tipo di scolatura
LD TR0
@AND CmdScolaggioNormale
MOV(021) &1 tempSotScola  ; Tipo di scolatura
LD TR0
SET nuovaSottorigaReq
; rung 12
@LD nuovaSottorigaReq
MOV(021) &2 tempSotStato
; rung 13
JME(005) #101

### Section scritturaSottoriga

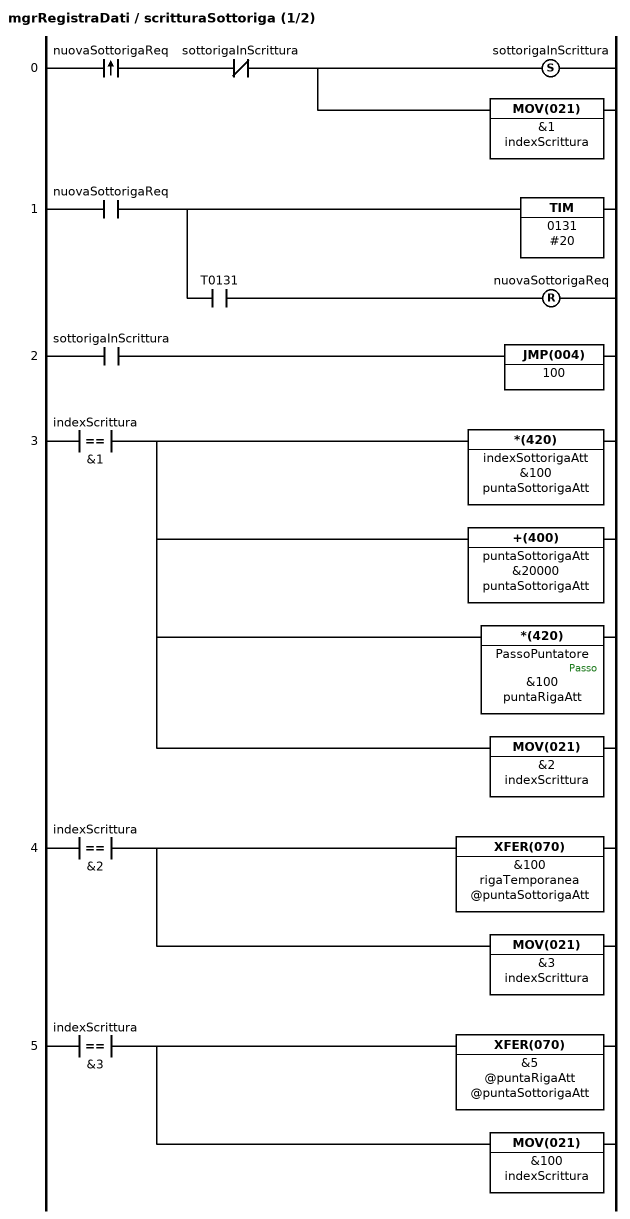
; rung 0
@LD nuovaSottorigaReq
ANDNOT sottorigaInScrittura
SET sottorigaInScrittura
MOV(021) &1 indexScrittura
; rung 1
LD nuovaSottorigaReq
TIM 0131 #20
AND T0131
RSET nuovaSottorigaReq
; rung 2
LD sottorigaInScrittura
JMP(004) 100
; rung 3
LD=(300) indexScrittura &1
*(420) indexSottorigaAtt &100 puntaSottorigaAtt
+(400) puntaSottorigaAtt &20000 puntaSottorigaAtt
*(420) PassoPuntatore &100 puntaRigaAtt  ; Passo
MOV(021) &2 indexScrittura
; rung 4
LD=(300) indexScrittura &2
XFER(070) &100 rigaTemporanea @puntaSottorigaAtt
MOV(021) &3 indexScrittura
; rung 5
LD=(300) indexScrittura &3
XFER(070) &5 @puntaRigaAtt @puntaSottorigaAtt
MOV(021) &100 indexScrittura

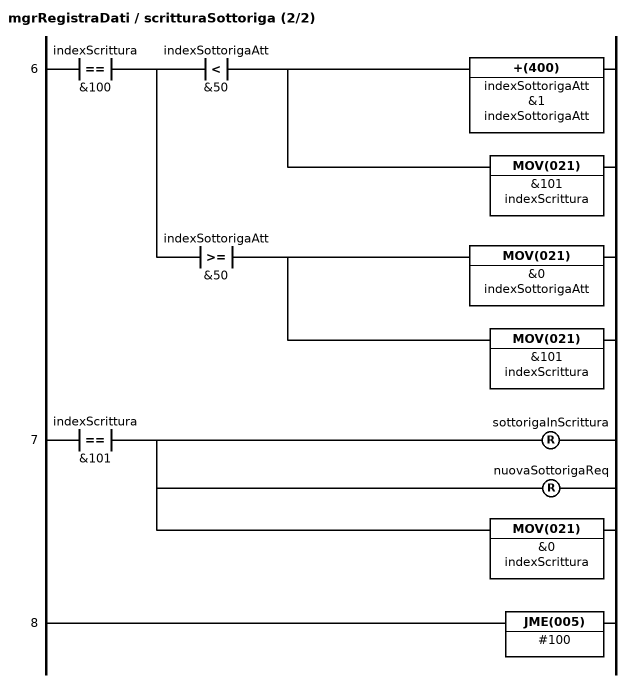
; rung 6
LD=(300) indexScrittura &100
OUT TR0
AND<(310) indexSottorigaAtt &50
+(400) indexSottorigaAtt &1 indexSottorigaAtt
MOV(021) &101 indexScrittura
LD TR0
AND>=(325) indexSottorigaAtt &50
MOV(021) &0 indexSottorigaAtt
MOV(021) &101 indexScrittura
; rung 7
LD=(300) indexScrittura &101
RSET sottorigaInScrittura
RSET nuovaSottorigaReq
MOV(021) &0 indexScrittura
; rung 8
JME(005) #100

### Section END
; rung 0
END(001)